(* IEC 61131-3 sources: plcassist-cli/packages/volt-lsp-iec/test-corpus/pro2193/Device/Plc Logic/Application/99 Library/Function Blocks/Actuators/Safety Gates, 6 files *)

(* ---- ISafetyGate.itf ---- *)
INTERFACE ISafetyGate
EXTENDS __SYSTEM.IQueryInterface

{attribute 'monitoring':='call'}
PROPERTY PUBLIC GateState : enumGateStates
GET
END_GET
END_PROPERTY

{attribute 'monitoring':='call'}
PROPERTY PUBLIC LockButtonPushed : BOOL
GET
END_GET
END_PROPERTY

END_INTERFACE

(* ---- GateBaseFB.fb ---- *)
{attribute 'symbol' := 'none'}
{attribute 'monitoring_display' := 'eState'}
FUNCTION_BLOCK PUBLIC ABSTRACT GateBaseFB
EXTENDS ModuleRegisterableFB
IMPLEMENTS ISafetyGate
VAR_INPUT
	xSafetyGateClosed			: BOOL;				// Input from safety sensor
	ButtonLock					: PushButtonLedFB;	// Button Request gate lock
	ButtonUnLock				: PushButtonLedFB;	// Button Request gate unlock
	xAcknowledge				: BOOL;				// Input from safety relay
	xGateAllowedOpen			: BOOL;				// High when it is allowed to open the gate (Stopped or Idle state)
	xGateAllowedClosed			: BOOL	:= TRUE;	// High when it is allowed to close the gate (System.Off)

	xIMMGateClose				: BOOL	:= TRUE;	// Input from IMM gate closed	(TRUE when in use without IMM)
	xGateAllowedOpenIMM			: BOOL	:= TRUE;	// In case of Euromap 78		(TRUE when in use without IMM)

	xRequestForOpening			: REFERENCE TO BOOL;	// Request for opening
	xAcknowledgement			: REFERENCE TO BOOL;	// Request for acknowledgement

	moduleThatBlocks			: IModuleBlocksSafetyGate;
END_VAR
VAR
	GateOutput					: ActuatorFB;		// Magnet or Pneumatic

	{attribute 'symbol' := 'read'}	eState						: enumGateStates;

	GateOpenedAlarm				: SetErrorFB;
END_VAR
VAR_STAT
	// ONLY USE DURING TESTING AT BRINK!
	// ONLY USE WHEN YOU ARE NEXT TO THE MACHINE AND CAN VISUALLY CHECK IF MACHINE IS EMPTY!
	acknowledgeAllGates			: BOOL;		// Acknowledge all gates for the machine
END_VAR

SUPER^();

CASE eState OF
	enumGateStates.Opened:
		ButtonUnLock.Flash();
		ButtonLock.Off();

	enumGateStates.Closed:
		IF GateOutput.Map() THEN		// Gate is locked, but some other gate is still open
			ButtonUnLock.Solid();
			ButtonLock.SetOrReset(GlobalVars.BlinkerPulseSlow);
		ELSIF xGateAllowedClosed THEN	// Gate is open and able to close
			ButtonUnLock.Solid();
			ButtonLock.Flash();
		ELSE							// Gate is not allowed to close
			ButtonUnLock.SetOrReset(GlobalVars.BlinkerPulseFast);
			ButtonLock.SetOrReset(GlobalVars.BlinkerPulseFast);
		END_IF

	enumGateStates.Acknowledged:
		ButtonUnLock.Solid();
		ButtonLock.Off();

	enumGateStates.Locked:
		ButtonUnLock.Off();
		ButtonLock.Off();
END_CASE

GateOutput();
ButtonLock();
ButtonUnLock();

IF __ISVALIDREF(xRequestForOpening) THEN
	xRequestForOpening	S= ButtonUnLock.buttonInput AND xGateAllowedOpen;
END_IF
IF __ISVALIDREF(xAcknowledgement) THEN
	xAcknowledgement	S= (ButtonLock.buttonInput OR acknowledgeAllGates) AND xSafetyGateClosed;
END_IF

GateOpenedAlarm(
	moduleHandler	:= ModuleHandler,
	textRefId		:= General_Unit_Errors,
	errorId			:= 5,
	alarmCondition	:= GateState = enumGateStates.Opened,
	alarmDelay		:= 0.0,
	severity		:= enumErrorSeverity.Information,
	reaction		:= enumErrorReaction.No_reaction,
	active			=> );

// Give command to some module to move into a safe position.
IF  moduleThatBlocks <> 0
AND eState <> enumGateStates.Locked
AND_THEN NOT moduleThatBlocks.InSafePosForGate
THEN
	IF ButtonUnLock.ButtonPushed THEN
		moduleThatBlocks.GateOpenRequested();
	END_IF
	IF ButtonUnLock.ButtonReleased THEN
		moduleThatBlocks.GateOpenCancelled();
	END_IF
END_IF

//acknowledgeAllGates	:= FALSE;

END_FUNCTION_BLOCK

METHOD PROTECTED Cyclic
VAR_INST
	T_SafetyGateClosed		: BTON;
END_VAR

//{warning 'todo: xGateAllowedOpen is 1 cycle laag wanneer ser state = Stopping ... ']}
CASE eState OF
	enumGateStates.Opened:		// Machine OFF and gate open
		IF T_SafetyGateClosed.Set(In := xSafetyGateClosed, Pt := 0.5) THEN
			T_SafetyGateClosed.Reset();
			eState	:= enumGateStates.Closed;
		END_IF

	enumGateStates.Closed:		// Machine OFF, gate is closed, not acknowledged and still able to open
		IF (ButtonLock.ButtonPushed OR acknowledgeAllGates)
		AND xGateAllowedClosed
		THEN
			GateOutput.Set();
		END_IF

		IF ButtonUnLock.buttonInput	// Do not look at ButtonPushed trigger here. Open the gate when button is being pushed when entering state
		AND xGateAllowedOpen
		AND xGateAllowedOpenIMM
		AND (moduleThatBlocks = 0 OR_ELSE moduleThatBlocks.InSafePosForGate)	// Gate is not safe to open. First a module must move to a safe spot.
		THEN
			GateOutput.Reset();
		END_IF

		IF NOT xSafetyGateClosed THEN
			GateOutput.Reset();
			eState	:= enumGateStates.Opened;
		ELSIF xIMMGateClose AND xAcknowledge AND GateOutput.Map() THEN
			eState	:= enumGateStates.Acknowledged;
		END_IF

	enumGateStates.Acknowledged:	// Machine OFF, gate is closed, acknowledged but still able to open
		IF NOT xSafetyGateClosed THEN
			GateOutput.Reset();
			eState	:= enumGateStates.Opened;
		ELSIF (ButtonUnLock.ButtonPushed AND xGateAllowedOpen AND xGateAllowedOpenIMM)
		OR NOT xIMMGateClose
		OR NOT xAcknowledge
		OR NOT GateOutput.Map()
		THEN
			eState	:= enumGateStates.Closed;
		ELSIF NOT xGateAllowedOpen THEN
			eState	:= enumGateStates.Locked;
		END_IF

	enumGateStates.Locked:		// Locked and not able to open
		IF NOT xSafetyGateClosed THEN
			eState	:= enumGateStates.Opened;
		ELSIF NOT GateOutput.Map() THEN
			eState	:= enumGateStates.Closed;
		ELSIF xGateAllowedOpen THEN
			eState	:= enumGateStates.Acknowledged;
		END_IF
END_CASE
END_METHOD

// Maps the actuator to the physical output
METHOD PUBLIC MapGate : BOOL
MapGate := GateOutput.Map();
END_METHOD

{attribute 'monitoring':='call'}
PROPERTY PUBLIC GateState : enumGateStates
GET
VAR
END_VAR
GateState := eState;
END_GET
END_PROPERTY

{attribute 'monitoring' := 'call'}
PROPERTY LockButtonPushed : BOOL
GET
VAR
END_VAR
LockButtonPushed := ButtonLock.ButtonPushed OR acknowledgeAllGates;
END_GET
END_PROPERTY

(* ---- GateMagnetFB.fb ---- *)
{attribute 'symbol' := 'none'}
{attribute 'monitoring_display' := 'eState'}
FUNCTION_BLOCK GateMagnetFB
EXTENDS GateBaseFB
VAR
END_VAR

SUPER^();

END_FUNCTION_BLOCK

(* ---- GatePneumaticDrawerFB.fb ---- *)
{attribute 'symbol' := 'none'}
{attribute 'monitoring_display' := 'eState'}
FUNCTION_BLOCK GatePneumaticDrawerFB
EXTENDS GateBaseFB
VAR_INPUT
	drawer					: IModuleBlocksSafetyGate;
END_VAR
VAR
END_VAR

SUPER^();

END_FUNCTION_BLOCK

METHOD PROTECTED Cyclic
VAR_INST
	drawerLockedForGate	: BOOL;
	gateOpenPermission	: BOOL;
	Blinker				: BLINK;
END_VAR
SUPER^.Cyclic();

// Get drawer hardware control and prevent other actions on the drawer
IF  eState <> enumGateStates.Locked
AND (ButtonLock.buttonInput OR ButtonUnLock.buttonInput)
AND_THEN drawer.LockRequest(InstanceName)
THEN
	drawerLockedForGate := TRUE;
END_IF

IF (ButtonLock.buttonInput OR ButtonUnLock.buttonInput)					// Some button is being pressed
AND drawerLockedForGate													// Don't do anything when the drawer is not ours
AND (moduleThatBlocks = 0 OR_ELSE moduleThatBlocks.InSafePosForGate)	// Gate is not safe to open. First a module must move to a safe spot.
THEN
	// Drawers are a little different for every machine, so you can adjust how strong the cylinder acts here.
	Blinker(ENABLE:= TRUE, TIMELOW:= T#500MS, TIMEHIGH:= T#1500MS, OUT=> );
	IF drawer.InSafePosForGate OR Blinker.OUT THEN	// Cylinder must be set when on the safety sensor or on the high time of the blinker
		IF ButtonUnLock.buttonInput THEN
			drawer.GateOpenRequested();				// Help opening the gate
		ELSIF ButtonLock.buttonInput AND xGateAllowedClosed THEN
			drawer.GateCloseRequested();			// Help closing the gate
		END_IF
	ELSE
		drawer.GateOpenCancelled();					// Not in safe pos and blinker is low, or Button is released
		drawer.GateCloseCancelled();				// Not in safe pos and blinker is low, or Button is released
	END_IF
END_IF

IF (ButtonLock.ButtonReleased OR ButtonUnLock.ButtonReleased)
AND drawerLockedForGate
THEN
	drawerLockedForGate := FALSE;
	drawer.GateOpenCancelled();
	drawer.GateCloseCancelled();
	drawer.LockRelease(InstanceName);
END_IF
END_METHOD

(* ---- GatePneumaticFB.fb ---- *)
{attribute 'symbol' := 'none'}
{attribute 'monitoring_display' := 'eState'}
FUNCTION_BLOCK GatePneumaticFB
EXTENDS GateBaseFB
VAR
	AssistOpenGate			: ActuatorFB;
	AssistCloseGate			: ActuatorFB;
	AssistUnlock			: ActuatorFB;
END_VAR

SUPER^();

END_FUNCTION_BLOCK

METHOD PROTECTED Cyclic
VAR_INST
	T_DoorCloseAssist		: BTON;
	T_DoorOpenAssist		: BTON;
END_VAR
SUPER^.Cyclic();

AssistOpenGate();
AssistCloseGate();

AssistUnlock();
AssistUnlock.SetOrReset(AssistOpenGate.Map() OR AssistCloseGate.Map());

AssistOpenGate.Reset();
AssistCloseGate.Reset();

IF moduleThatBlocks <> 0 AND_THEN NOT moduleThatBlocks.InSafePosForGate THEN
	RETURN;
END_IF

IF T_DoorOpenAssist.Set(In := ButtonUnLock.buttonInput AND xGateAllowedOpen AND xGateAllowedOpenIMM, 0.5) THEN
	IF xSafetyGateClosed THEN
		AssistOpenGate.Set();
	ELSE
		AssistOpenGate.SetOrReset(GlobalVars.BlinkerNormal);
	END_IF
	AssistCloseGate.Reset();
ELSIF T_DoorCloseAssist.Set(In := ButtonLock.buttonInput AND xGateAllowedClosed, 0.5) THEN
	AssistOpenGate.Reset();
	IF xSafetyGateClosed THEN
		AssistCloseGate.Set();
	ELSE
		AssistCloseGate.SetOrReset(GlobalVars.BlinkerNormal);
	END_IF
END_IF
END_METHOD

// Maps the actuator to the physical output
METHOD PUBLIC MapAssistCloseGate : BOOL
MapAssistCloseGate := AssistCloseGate.Map();
END_METHOD

// Maps the actuator to the physical output
METHOD PUBLIC MapAssistOpenGate : BOOL
MapAssistOpenGate := AssistOpenGate.Map();
END_METHOD

// Maps the actuator to the physical output
METHOD PUBLIC MapAssistUnlock : BOOL
MapAssistUnlock := AssistUnlock.Map();
END_METHOD

(* ---- GatesControlIMMCircuitFB.fb ---- *)
{attribute 'monitoring_display' := 'GateStatus'}
FUNCTION_BLOCK GatesControlIMMCircuitFB
VAR_INPUT
	xGateAllowedOpen			: BOOL;				// High when it is allowed to open the gate (Stopped or Idle state)
	xSafetyGateRelay			: BOOL;
END_VAR
VAR_OUTPUT
	xPnozMulti2Acknowledgement	: BOOL;
END_VAR
VAR_IN_OUT
	xRequestForOpening			: BOOL;
	xAcknowledgement			: BOOL;
END_VAR
VAR
	IMMRequestForOpening		: ActuatorFB;
	IMMAcknowledgement			: ActuatorFB;
	Tr_AcknowledgementRequest	: R_Trig;
	T_SafetyGateRelay			: BTON;
	T_Timer						: BTON;
	GateStatus					: enumGateStates;
END_VAR

Tr_AcknowledgementRequest(CLK := xAcknowledgement);
T_SafetyGateRelay.Set(xSafetyGateRelay, 0.5);

CASE GateStatus OF
enumGateStates.Opened://Gate opened
	IMMRequestForOpening.SetOrReset(xGateAllowedOpen AND xRequestForOpening);
	IMMAcknowledgement.Reset();
	xPnozMulti2Acknowledgement	:= FALSE;

	IF xAcknowledgement AND NOT xRequestForOpening THEN
		GateStatus	:= enumGateStates.Closed;
	END_IF

enumGateStates.Closed://Gate closed and button pressed, Acknowledge request to PnozMulti2, IMM gate opened
	IMMRequestForOpening.Reset();
	IMMAcknowledgement.Reset();
	xPnozMulti2Acknowledgement	:= TRUE;
	T_Timer.Set(TRUE, 2);

	IF xSafetyGateRelay THEN
		T_Timer.Reset();
		GateStatus	:= enumGateStates.Acknowledged;
	ELSIF xRequestForOpening OR (T_Timer.Q AND NOT xAcknowledgement) THEN
		T_Timer.Reset();
		GateStatus	:= enumGateStates.Opened;
	END_IF

enumGateStates.Acknowledged://Gate Acknowledged, delay Acknowledge sinal to IMM
	IMMRequestForOpening.Reset();
	IMMAcknowledgement.Reset();
	xPnozMulti2Acknowledgement	:= FALSE;
	T_Timer.Set(TRUE, 0.1);

	IF T_SafetyGateRelay.Q AND T_Timer.Q THEN
		T_Timer.Reset();
		GateStatus	:= enumGateStates.Locked;
	ELSIF xRequestForOpening OR NOT xSafetyGateRelay THEN
		T_Timer.Reset();
		GateStatus	:= enumGateStates.Opened;
	END_IF

enumGateStates.Locked://Acknowledge signal to IMM for 0.5 second or Button is pressed
	IMMRequestForOpening.Reset();
	IMMAcknowledgement.SetOrReset(NOT T_Timer.Set(TRUE, 0.5) OR xAcknowledgement);
	xPnozMulti2Acknowledgement	:= xAcknowledgement;

	IF Tr_AcknowledgementRequest.Q THEN
		T_Timer.Reset();
		GateStatus	:= enumGateStates.Acknowledged;
	ELSIF xRequestForOpening OR NOT xSafetyGateRelay THEN
		T_Timer.Reset();
		GateStatus	:= enumGateStates.Opened;
	END_IF
END_CASE

xRequestForOpening	:= FALSE;
xAcknowledgement	:= FALSE;

IMMRequestForOpening();
IMMAcknowledgement();

END_FUNCTION_BLOCK
